INTERFACE I_ValueReader

METHOD ValueReader : HRESULT
VAR_IN_OUT
    stBuffer : ST_Span;
    stState  : ST_ParserInternalState;
END_VAR
VAR_OUTPUT
    anyOut : T_Any;
END_VAR
END_METHOD

END_INTERFACE

(* stored: Version 1.1.0.1
   Itf I_ValueReader: Id {37fdf320-e2a9-4052-bfd4-6be9bb2582e7}
   Method ValueReader: Id {3b7eefb9-456c-4f6e-87f8-51b5178c58ba} *)
